KUKA KRL program: e_fraes2.src, e_fraes2.dat

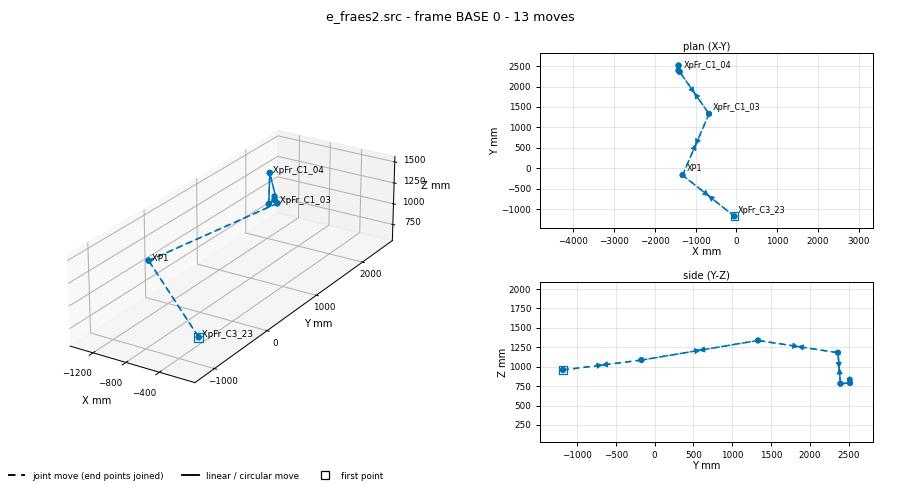
[picture p0: tool path of e_fraes2.src in frame BASE 0, 13 of 13 moves have a stored position in this frame; points joined in program order, loops and branches not executed]
--- e_fraes2.src ---
&ACCESS RVP3
&REL 3
&COMMENT INI Dress C1
&PARAM DISKPATH = KRC:\R1\Program
&PARAM TEMPLATE = C:\KRC\Roboter\Template\vorgabe
&PARAM EDITMASK = *
DEF e_fraes2( )
;FOLD INI
  ;FOLD BASISTECH INI
    GLOBAL INTERRUPT DECL 3 WHEN $STOPMESS==TRUE DO IR_STOPM ( )
    INTERRUPT ON 3
    BAS (#INITMOV,0 )
  ;ENDFOLD (BASISTECH INI)
;FOLD SPOTTECH INI
USERSPOT(#INIT)

;ENDFOLD (SPOTTECH INI)
;FOLD GRIPPERTECH INI
USER_GRP(0,DUMMY,DUMMY,GDEFAULT)
;ENDFOLD (GRIPPERTECH INI)
  ;FOLD USER INI
    ;Make your modifications here

  ;ENDFOLD (USER INI)
;ENDFOLD (INI)

; Caracterização dos meios de produção:
; Versão Atual:08/09/2015
; Name: P13.050-R2 CHANGES: Fresa C1
; (F2 6640 0018 984)



chk_w2_wechs_ok ( )    ; CHECK TOOL C1


;FOLD PTP pFr_C3_23 CONT Vel=100 % PDAT21 Tool[2]:Gun C1 Base[0];%{PE}%R 8.2.20,%MKUKATPBASIS,%CMOVE,%VPTP,%P 1:PTP, 2:pFr_C3_23, 3:C_DIS, 5:100, 7:PDAT21
$BWDSTART=FALSE
PDAT_ACT=PPDAT21
FDAT_ACT=FpFr_C3_23
BAS(#PTP_PARAMS,100)
PTP XpFr_C3_23 C_DIS
;ENDFOLD

;FOLD PTP P1 CONT Vel=100 % PDAT22 Tool[2]:Gun C1 Base[0];%{PE}%R 8.2.20,%MKUKATPBASIS,%CMOVE,%VPTP,%P 1:PTP, 2:P1, 3:C_DIS, 5:100, 7:PDAT22
$BWDSTART=FALSE
PDAT_ACT=PPDAT22
FDAT_ACT=FP1
BAS(#PTP_PARAMS,100)
PTP XP1 C_DIS
;ENDFOLD
;FOLD PTP pFr_C1_03 CONT Vel=100 % PDAT3 Tool[2]:Gun C1 Base[0];%{PE}%R 8.2.20,%MKUKATPBASIS,%CMOVE,%VPTP,%P 1:PTP, 2:pFr_C1_03, 3:C_DIS, 5:100, 7:PDAT3
$BWDSTART=FALSE
PDAT_ACT=PPDAT3
FDAT_ACT=FpFr_C1_03
BAS(#PTP_PARAMS,100)
PTP XpFr_C1_03 C_DIS
;ENDFOLD
;FOLD PTP pFr_C1_04 CONT Vel=100 % PDAT2 Tool[2]:Gun C1 Base[0];%{PE}%R 8.2.20,%MKUKATPBASIS,%CMOVE,%VPTP,%P 1:PTP, 2:pFr_C1_04, 3:C_DIS, 5:100, 7:PDAT2
$BWDSTART=FALSE
PDAT_ACT=PPDAT2
FDAT_ACT=FpFr_C1_04
BAS(#PTP_PARAMS,100)
PTP XpFr_C1_04 C_DIS
;ENDFOLD

;FOLD LIN P3 CONT Vel=1 m/s CPDAT2 Tool[2]:Gun C1 Base[0];%{PE}%R 8.2.20,%MKUKATPBASIS,%CMOVE,%VLIN,%P 1:LIN, 2:P3, 3:C_DIS C_DIS, 5:1, 7:CPDAT2
$BWDSTART=FALSE
LDAT_ACT=LCPDAT2
FDAT_ACT=FP3
BAS(#CP_PARAMS,1)
LIN XP3 C_DIS C_DIS
;ENDFOLD
;FOLD LIN pFr_C1_06 CONT Vel=1 m/s CPDAT1 Tool[2]:Gun C1 Base[0];%{PE}%R 8.2.20,%MKUKATPBASIS,%CMOVE,%VLIN,%P 1:LIN, 2:pFr_C1_06, 3:C_DIS C_DIS, 5:1, 7:CPDAT1
$BWDSTART=FALSE
LDAT_ACT=LCPDAT1
FDAT_ACT=FpFr_C1_06
BAS(#CP_PARAMS,1)
LIN XpFr_C1_06 C_DIS C_DIS
;ENDFOLD

;FOLD ; Ponto de fresagem;%{PE}%R 8.2.20,%MKUKATPBASIS,%CCOMMENT,%VNORMAL,%P 2:Ponto  de  fresagem
;ENDFOLD
;FOLD TIP.LIN_ Dress4, Spot Gun 1 , RETR open , Tool[2], Base[0], EXT.TCP=FALSE;%{PE}%MKUKATPUSER
FDAT_ACT=FDress4
BAS(#FRAMES)
LIN  XDress4
S_ACT.GUN=1
S_ACT.RETR=#opn
S_READY=FALSE
USERSPOT (#DRESS,S_ACT )
WAIT FOR  S_READY
;ENDFOLD

;FOLD LIN pFr_C1_08 Vel=1 m/s CPDAT3 Tool[2]:Gun C1 Base[0];%{PE}%R 8.2.20,%MKUKATPBASIS,%CMOVE,%VLIN,%P 1:LIN, 2:pFr_C1_08, 3:, 5:1, 7:CPDAT3
$BWDSTART=FALSE
LDAT_ACT=LCPDAT3
FDAT_ACT=FpFr_C1_08
BAS(#CP_PARAMS,1)
LIN XpFr_C1_08
;ENDFOLD
;FOLD LIN P4 CONT Vel=1 m/s CPDAT4 Tool[2]:Gun C1 Base[0];%{PE}%R 8.2.20,%MKUKATPBASIS,%CMOVE,%VLIN,%P 1:LIN, 2:P4, 3:C_DIS C_DIS, 5:1, 7:CPDAT4
$BWDSTART=FALSE
LDAT_ACT=LCPDAT4
FDAT_ACT=FP4
BAS(#CP_PARAMS,1)
LIN XP4 C_DIS C_DIS
;ENDFOLD

;FOLD PTP pFr_C1_15 PDAT13 SPOT Gun=1 RETR OPN PgNo1=251 ACTIVE=1 Tool[2]:Gun C1 Base[0];%{PE}%R 8.2.2,%MKUKATPSPOT,%CSPOT,%VPTP,%P 1:PTP, 2:pFr_C1_15, 3:, 5:100, 7:PDAT13, 10:1, 12:#FIRST, 14:#OPN, 16:251, 18:1, 20:0, 22:0, 24:1, 25:NORMAL
$BWDSTART=FALSE
PDAT_ACT=PPDAT13
FDAT_ACT=FpFr_C1_15
BAS(#PTP_PARAMS,PPDAT13.VEL)
S_ACT.GUN=1
S_ACT.PAIR=SDEFAULT.PAIR
S_ACT.RETR=#OPN
S_ACT.CLO_TM=1
S_ACT.PGNO1=251
S_ACT.PGNO2=SDEFAULT.PGNO2
S_ACT.PRESS1=SDEFAULT.PRESS1
S_ACT.PRESS2=SDEFAULT.PRESS2
S_READY=FALSE
PTP XpFr_C1_15
USERSPOT(#SPOT, S_ACT)
WAIT FOR S_READY
;ENDFOLD
;FOLD PTP pFr_C1_18 CONT Vel=100 % PDAT16 Tool[2]:Gun C1 Base[0];%{PE}%R 8.2.20,%MKUKATPBASIS,%CMOVE,%VPTP,%P 1:PTP, 2:pFr_C1_18, 3:C_DIS, 5:100, 7:PDAT16
$BWDSTART=FALSE
PDAT_ACT=PPDAT16
FDAT_ACT=FpFr_C1_18
BAS(#PTP_PARAMS,100)
PTP XpFr_C1_18 C_DIS
;ENDFOLD
;FOLD PTP P2 CONT Vel=100 % PDAT23 Tool[2]:Gun C1 Base[0];%{PE}%R 8.2.20,%MKUKATPBASIS,%CMOVE,%VPTP,%P 1:PTP, 2:P2, 3:C_DIS, 5:100, 7:PDAT23
$BWDSTART=FALSE
PDAT_ACT=PPDAT23
FDAT_ACT=FP2
BAS(#PTP_PARAMS,100)
PTP XP2 C_DIS
;ENDFOLD
;FOLD PTP pFr_C1_21 CONT Vel=100 % PDAT19 Tool[2]:Gun C1 Base[0];%{PE}%R 8.2.20,%MKUKATPBASIS,%CMOVE,%VPTP,%P 1:PTP, 2:pFr_C1_21, 3:C_DIS, 5:100, 7:PDAT19
$BWDSTART=FALSE
PDAT_ACT=PPDAT19
FDAT_ACT=FpFr_C1_21
BAS(#PTP_PARAMS,100)
PTP XpFr_C1_21 C_DIS
;ENDFOLD

END

--- e_fraes2.dat ---
&ACCESS RVP3
&REL 3
&COMMENT INI Dress C1
&PARAM DISKPATH = KRC:\R1\Program
&PARAM TEMPLATE = C:\KRC\Roboter\Template\vorgabe
&PARAM EDITMASK = *
DEFDAT  e_fraes2
;FOLD EXTERNAL DECLARATIONS;%{PE}%MKUKATPBASIS,%CEXT,%VCOMMON,%P
;FOLD GRIPPERTECH EXT
EXT  H50 (INT  :IN,INT  :IN,INT  :IN,GRP_TYP  :IN )
;ENDFOLD (GRIPPERTECH EXT)
;FOLD SPOTTECH EXT
EXT  USERSPOT (S_COMMAND  :IN,SPOT_TYPE  :IN )
;ENDFOLD (SPOTTECH EXT)
;FOLD BASISTECH EXT;%{PE}%MKUKATPBASIS,%CEXT,%VEXT,%P
EXT  BAS (BAS_COMMAND  :IN,REAL  :IN )
DECL INT SUCCESS
;ENDFOLD (BASISTECH EXT)
;FOLD USER EXT;%{E}%MKUKATPUSER,%CEXT,%VEXT,%P
;Make your modifications here

;ENDFOLD (USER EXT)
;ENDFOLD (EXTERNAL DECLARATIONS)
DECL BASIS_SUGG_T LAST_BASIS={POINT1[] "P5                      ",POINT2[] "P5                      ",CP_PARAMS[] "CPDAT0                  ",PTP_PARAMS[] "PDAT1                   ",CONT[] "                        ",CP_VEL[] "2.0                     ",PTP_VEL[] "100                     ",SYNC_PARAMS[] "SYNCDAT                 ",SPL_NAME[] "S0                      "}
DECL PDAT PPDAT2={VEL 100.0,ACC 100.0,APO_DIST 100.0,APO_MODE #CDIS}
DECL PDAT PPDAT3={VEL 100.0,ACC 100.0,APO_DIST 100.0,APO_MODE #CDIS}
DECL LDAT LCPDAT1={VEL 2.0,ACC 100.0,APO_DIST 100.0,APO_FAC 50.0,AXIS_VEL 100.0,AXIS_ACC 100.0,ORI_TYP #VAR,CIRC_TYP #BASE,JERK_FAC 50.0,GEAR_JERK 50.0,EXAX_IGN 0}
DECL LDAT LCPDAT3={VEL 2.0,ACC 100.0,APO_DIST 100.0,APO_FAC 50.0,AXIS_VEL 100.0,AXIS_ACC 100.0,ORI_TYP #VAR,CIRC_TYP #BASE,JERK_FAC 50.0,GEAR_JERK 50.0,EXAX_IGN 0}
DECL FDAT FDress4={TOOL_NO 2,BASE_NO 0,IPO_FRAME #BASE}
DECL E6POS XDress4={X -1416.16199,Y 2511.43506,Z 835.319275,A 89.5502472,B -4.12478209,C 1.33925104,S 2,T 2,E1 197.747192,E2 0.0,E3 0.0,E4 0.0,E5 0.0,E6 0.0}
DECL SPOT_SUGG_T LAST_SPOT={GUN[] "3                       ",RETR_CMD[] "#OPN                    ",CHOISE[] "#FIRST                  ",CLO_TM[] "1                       ",PGNO1[] "1                       ",PRESS1[] "0                       ",PGNO2[] "1                       ",PRESS2[] "0                       ",SPOT_PARAMS[] "NORMAL                  "}
DECL PDAT PPDAT13={VEL 100.0,ACC 100.0,APO_DIST 100.0}
DECL PDAT PPDAT16={VEL 100.0,ACC 100.0,APO_DIST 100.0,APO_MODE #CDIS}
DECL PDAT PPDAT19={VEL 100.0,ACC 100.0,APO_DIST 100.0,APO_MODE #CDIS}
DECL E6POS XpFr_C1_03={X -670.706177,Y 1330.34497,Z 1337.745,A 103.089897,B -6.77851582,C 2.15911889,S 2,T 10,E1 196.484695,E2 0.0,E3 0.0,E4 0.0,E5 0.0,E6 0.0}
DECL FDAT FpFr_C1_03={TOOL_NO 2,BASE_NO 0,IPO_FRAME #BASE,POINT2[] " ",TQ_STATE FALSE}
DECL E6POS XpFr_C1_04={X -1389.47498,Y 2359.5459,Z 1180.46204,A 89.5501785,B -4.12478781,C 1.33930099,S 2,T 2,E1 197.747803,E2 0.0,E3 0.0,E4 0.0,E5 0.0,E6 0.0}
DECL FDAT FpFr_C1_04={TOOL_NO 2,BASE_NO 0,IPO_FRAME #BASE,POINT2[] " ",TQ_STATE FALSE}
DECL E6POS XpFr_C1_06={X -1417.18506,Y 2514.66895,Z 790.570618,A 89.5503006,B -4.1247611,C 1.33920801,S 2,T 2,E1 197.747101,E2 0.0,E3 0.0,E4 0.0,E5 0.0,E6 0.0}
DECL FDAT FpFr_C1_06={TOOL_NO 2,BASE_NO 0,IPO_FRAME #BASE,POINT2[] " ",TQ_STATE FALSE}
DECL E6POS XpFr_C1_08={X -1417.18506,Y 2514.66895,Z 790.570618,A 89.5501633,B -4.12477303,C 1.33921599,S 2,T 2,E1 197.747101,E2 0.0,E3 0.0,E4 0.0,E5 0.0,E6 0.0}
DECL FDAT FpFr_C1_08={TOOL_NO 2,BASE_NO 0,IPO_FRAME #BASE,POINT2[] " ",TQ_STATE FALSE}
DECL E6POS XpFr_C1_15={X -1389.47498,Y 2359.5459,Z 1180.46204,A 89.5501785,B -4.12478781,C 1.33930099,S 2,T 2,E1 197.747803,E2 0.0,E3 0.0,E4 0.0,E5 0.0,E6 0.0}
DECL FDAT FpFr_C1_15={TOOL_NO 2,BASE_NO 0,IPO_FRAME #BASE,POINT2[] " ",TQ_STATE FALSE}
DECL E6POS XpFr_C1_18={X -670.706177,Y 1330.34497,Z 1337.745,A 103.089897,B -6.77851582,C 2.15911889,S 2,T 10,E1 196.484695,E2 0.0,E3 0.0,E4 0.0,E5 0.0,E6 0.0}
DECL FDAT FpFr_C1_18={TOOL_NO 2,BASE_NO 0,IPO_FRAME #BASE,POINT2[] " ",TQ_STATE FALSE}
DECL E6POS XpFr_C1_21={X -47.513031,Y -1179.89001,Z 958.025391,A -84.9619904,B -3.94106507,C -0.446948111,S 2,T 10,E1 197.230392,E2 0.0,E3 0.0,E4 0.0,E5 0.0,E6 0.0}
DECL FDAT FpFr_C1_21={TOOL_NO 2,BASE_NO 0,IPO_FRAME #BASE,POINT2[] " ",TQ_STATE FALSE}
DECL E6POS XPFR_C3_23={X -47.5121689,Y -1179.89502,Z 958.024475,A -84.9614716,B -3.94118309,C -0.447002709,S 2,T 10,E1 197.230103,E2 0.0,E3 0.0,E4 0.0,E5 0.0,E6 0.0}
DECL FDAT FpFr_C3_23={TOOL_NO 2,BASE_NO 0,IPO_FRAME #BASE,POINT2[] " ",TQ_STATE FALSE}
DECL PDAT PPDAT21={VEL 100.0,ACC 100.0,APO_DIST 100.0,APO_MODE #CDIS}
DECL E6POS XP1={X -1319.37903,Y -170.242096,Z 1085.29797,A -157.389603,B -13.8282804,C -1.68598902,S 2,T 10,E1 195.473007,E2 0.0,E3 0.0,E4 0.0,E5 0.0,E6 0.0}
DECL FDAT FP1={TOOL_NO 2,BASE_NO 0,IPO_FRAME #BASE,POINT2[] " ",TQ_STATE FALSE}
DECL PDAT PPDAT22={VEL 100.0,ACC 100.0,APO_DIST 100.0,APO_MODE #CDIS}
DECL E6POS XP2={X -1319.37903,Y -170.241806,Z 1085.29797,A -157.389496,B -13.82827,C -1.68599999,S 2,T 10,E1 195.473206,E2 0.0,E3 0.0,E4 0.0,E5 0.0,E6 0.0}
DECL FDAT FP2={TOOL_NO 2,BASE_NO 0,IPO_FRAME #BASE,POINT2[] " ",TQ_STATE FALSE}
DECL PDAT PPDAT23={VEL 100.0,ACC 100.0,APO_DIST 100.0,APO_MODE #CDIS}
DECL E6POS XP3={X -1418.15405,Y 2391.30493,Z 781.675171,A 89.5501328,B -4.1247592,C 1.33922601,S 2,T 2,E1 197.747406,E2 0.0,E3 0.0,E4 0.0,E5 0.0,E6 0.0}
DECL FDAT FP3={TOOL_NO 2,BASE_NO 0,IPO_FRAME #BASE,POINT2[] " ",TQ_STATE FALSE}
DECL LDAT LCPDAT2={VEL 2.0,ACC 100.0,APO_DIST 100.0,APO_FAC 50.0,AXIS_VEL 100.0,AXIS_ACC 100.0,ORI_TYP #VAR,CIRC_TYP #BASE,JERK_FAC 50.0,GEAR_JERK 50.0,EXAX_IGN 0}
DECL E6POS XP4={X -1418.15295,Y 2391.30493,Z 781.674927,A 89.550148,B -4.12475014,C 1.33920002,S 2,T 2,E1 197.747406,E2 0.0,E3 0.0,E4 0.0,E5 0.0,E6 0.0}
DECL FDAT FP4={TOOL_NO 2,BASE_NO 0,IPO_FRAME #BASE,POINT2[] " ",TQ_STATE FALSE}
DECL LDAT LCPDAT4={VEL 2.0,ACC 100.0,APO_DIST 100.0,APO_FAC 50.0,AXIS_VEL 100.0,AXIS_ACC 100.0,ORI_TYP #VAR,CIRC_TYP #BASE,JERK_FAC 50.0,GEAR_JERK 50.0,EXAX_IGN 0}
DECL E6POS XP5={X -1416.16394,Y 2511.42993,Z 835.316528,A 89.550621,B -4.12446499,C 1.33943295,S 2,T 2,E1 197.747604,E2 0.0,E3 0.0,E4 0.0,E5 0.0,E6 0.0}
DECL FDAT FP5={TOOL_NO 2,BASE_NO 0,IPO_FRAME #BASE,POINT2[] " ",TQ_STATE FALSE}
DECL PDAT PPDAT1={VEL 100.0,ACC 100.0,APO_DIST 100.0}
ENDDAT
